PROGRAM MAIN
VAR

	
END_VAR

loopCounter := loopCounter + 1;

PRG_ReadModbusSensorData();

(* PRG_HandleUserInputs(); *)

PRG_UpdateMotor();

//PRG_UpdateTemperatureControl();
PRG_BAT_TemperatureControl();

PRG_UpdatePressureSensor();
PRG_UpdateFlowRateSensor();
PRG_UpdatePhControl();
PRG_UpdateGasSupply();
PRG_UpdateRoomTempRh();
PRG_GasAnalysis();

END_PROGRAM

(* stored: Version 1.1.0.1, ProductVersion 3.1.4022.12
   POU MAIN: Id {6de127fa-b6f4-4656-b169-9e870eadfc1d}, SpecialFunc None *)
